{attribute 'qualified_only'}
VAR_GLOBAL CONSTANT
    stConfig : ST_MachinePreparationConfig := (
        // 托盘机构
        fTrayXStandby := -95.0,
        fTrayZStandby := -734.0,

        // 阻尼器上下料机构
        // 与当前工程FB_DamperProcess中的(1,1)坐标保持一致
        fDamperXStandby := -191.5,
        fDamperYStandby := 95.0,
        fDamperZStandby := 110.0,
        fDamperRotationZero := 0.0,

        // 转台机构
        fClampOpenPosition := 93.0,
        fTurntableZero := 10.5,

        // 螺丝刀机构
        fScrewdriverYZero := 0.0,
        fScrewdriverZSafe := 85.0,

        // 临时调试速度
        fTrayVelocity := 50.0,
        fDamperVelocity := 50.0,
        fDamperRotationVelocity := 30.0,
        fClampVelocity := 15.0,
        fTurntableVelocity := 60.0,
        fScrewdriverVelocity := 10.0,

        fLinearTolerance := 0.01,
        fRotationTolerance := 0.1,

        tReadyTimeout := T#15S,
        tMotionTimeout := T#60S
    );
END_VAR

(* stored: Version 1.1.0.1, ProductVersion 3.1.4026.20
   GVL GVL_MachinePreparation: Id {313d3776-b1fb-4c58-be7e-75adffd0555c} *)
